TYPE T_Capacity : DINT(0..2147483647); END_TYPE

(* stored: Version 1.1.0.1, ProductVersion 3.1.4024.4
   DUT T_Capacity: Id {6bb70770-25cb-0d37-0346-8c0e1840418d} *)
